LIN {X 0,Y 64.244,Z 442.937,A -85,B 0,C 180,E1 -28515.759,E2 -28515.759} C_VEL
LIN {X 0,Y 63.406,Z 448.254,A -85,B 0,C 180,E1 -28523.644,E2 -28523.644} C_VEL
LIN {X 0,Y 63.515,Z 451.726,A -85,B 0,C 180,E1 -28530.008,E2 -28530.008} C_VEL
LIN {X 0,Y 63.381,Z 454.429,A -85,B 0,C 180,E1 -28536.374,E2 -28536.374} C_VEL
LIN {X 0,Y 63.772,Z 456.467,A -85,B 0,C 180,E1 -28542.741,E2 -28542.741} C_VEL
LIN {X 0,Y 64.939,Z 458.028,A -85,B 0,C 180,E1 -28548.954,E2 -28548.954} C_VEL
LIN {X 0,Y 66.859,Z 459.178,A -85,B 0,C 180,E1 -28554.872,E2 -28554.872} C_VEL
LIN {X 0,Y 69.441,Z 459.905,A -85,B 0,C 180,E1 -28560.409,E2 -28560.409} C_VEL
LIN {X 0,Y 72.688,Z 460.091,A -85,B 0,C 180,E1 -28565.468,E2 -28565.468} C_VEL
LIN {X 0,Y 80.971,Z 459.289,A -85,B 0,C 180,E1 -28573.985,E2 -28573.985} C_VEL
LIN {X 0,Y 85.695,Z 458.239,A -85,B 0,C 180,E1 -28577.579,E2 -28577.579} C_VEL
LIN {X 0,Y 90.746,Z 456.64,A -85,B 0,C 180,E1 -28580.765,E2 -28580.765} C_VEL
LIN {X 0,Y 95.673,Z 454.631,A -85,B 0,C 180,E1 -28584.004,E2 -28584.004} C_VEL
LIN {X 0,Y 97.875,Z 453.563,A -85,B 0,C 180,E1 -28585.671,E2 -28585.671} C_VEL
LIN {X 0,Y 99.222,Z 452.513,A -85,B 0,C 180,E1 -28588.217,E2 -28588.217} C_VEL
LIN {X 0,Y 99.958,Z 451.651,A -85,B 0,C 180,E1 -28590.513,E2 -28590.513} C_VEL
LIN {X 0,Y 100.672,Z 450.423,A -85,B 0,C 180,E1 -28595.233,E2 -28595.233} C_VEL
LIN {X 0,Y 101.17,Z 449.63,A -85,B 0,C 180,E1 -28599.672,E2 -28599.672} C_VEL
LIN {X 0,Y 101.648,Z 449.123,A -85,B 0,C 180,E1 -28605.476,E2 -28605.476} C_VEL
LIN {X 0,Y 101.76,Z 449.101,A -85,B 0,C 180,E1 -28608.038,E2 -28608.038} C_VEL
LIN {X 0,Y 101.473,Z 449.465,A -85,B 0,C 180,E1 -28612.034,E2 -28612.034} C_VEL
LIN {X 0,Y 100.225,Z 450.423,A -85,B 0,C 180,E1 -28615.975,E2 -28615.975} C_VEL
LIN {X 0,Y 98.443,Z 451.251,A -85,B 0,C 180,E1 -28618.299,E2 -28618.299} C_VEL
LIN {X 0,Y 91.433,Z 453.624,A -85,B 0,C 180,E1 -28622.083,E2 -28622.083} C_VEL
LIN {X 0,Y 84.871,Z 455.149,A -85,B 0,C 180,E1 -28626.388,E2 -28626.388} C_VEL
LIN {X 0,Y 78.872,Z 455.858,A -85,B 0,C 180,E1 -28631.4,E2 -28631.4} C_VEL
LIN {X 0,Y 73.6,Z 455.754,A -85,B 0,C 180,E1 -28637.252,E2 -28637.252} C_VEL
LIN {X 0,Y 69.109,Z 454.82,A -85,B 0,C 180,E1 -28643.996,E2 -28643.996} C_VEL
LIN {X 0,Y 64.32,Z 451.791,A -85,B 0,C 180,E1 -28655.889,E2 -28655.889} C_VEL
LIN {X 0,Y 62.729,Z 448.38,A -85,B 0,C 180,E1 -28664.779,E2 -28664.779} C_VEL
LIN {X 0,Y 62.587,Z 443.781,A -85,B 0,C 180,E1 -28673.927,E2 -28673.927} C_VEL
LIN {X 0,Y 63.626,Z 438.495,A -85,B 0,C 180,E1 -28682.073,E2 -28682.073} C_VEL
LIN {X 0,Y 65.033,Z 433.873,A -85,B 0,C 180,E1 -28687.767,E2 -28687.767} C_VEL
LIN {X 0,Y 67.018,Z 428.034,A -85,B 0,C 180,E1 -28693.547,E2 -28693.547} C_VEL
LIN {X 0,Y 69.631,Z 420.592,A -85,B 0,C 180,E1 -28699.279,E2 -28699.279} C_VEL
LIN {X 0,Y 71.829,Z 414.232,A -85,B 0,C 180,E1 -28703.141,E2 -28703.141} C_VEL
LIN {X 0,Y 71.986,Z 407.933,A -85,B 0,C 180,E1 -28706.877,E2 -28706.877} C_VEL
LIN {X 0,Y 71.696,Z 402.285,A -85,B 0,C 180,E1 -28709.993,E2 -28709.993} C_VEL
LIN {X 0,Y 70.155,Z 394.65,A -85,B 0,C 180,E1 -28714.159,E2 -28714.159} C_VEL
LIN {X 0,Y 65.944,Z 385.726,A -85,B 0,C 180,E1 -28719.965,E2 -28719.965} C_VEL
LIN {X 0,Y 65.843,Z 385.09,A -85,B 0,C 180,E1 -28720.369,E2 -28720.369} C_VEL
LIN {X 0,Y 65.627,Z 385.123,A -85,B 0,C 180,E1 -28725.487,E2 -28725.487} C_VEL
LIN {X 0,Y 65.237,Z 385.169,A -85,B 0,C 180,E1 -28735.517,E2 -28735.517} C_VEL
LIN {X 0,Y 65.249,Z 385.167,A -85,B 0,C 180,E1 -28740.477,E2 -28740.477} C_VEL
LIN {X 0,Y 65.056,Z 385.207,A -85,B 0,C 180,E1 -28743.912,E2 -28743.912} C_VEL
LIN {X 0,Y 64.301,Z 385.311,A -85,B 0,C 180,E1 -28747.324,E2 -28747.324} C_VEL
LIN {X 0,Y 62.55,Z 385.533,A -85,B 0,C 180,E1 -28752.478,E2 -28752.478} C_VEL
LIN {X 0,Y 58.456,Z 386.017,A -85,B 0,C 180,E1 -28765.63,E2 -28765.63} C_VEL
LIN {X 0,Y 58.13,Z 386.048,A -85,B 0,C 180,E1 -28769.694,E2 -28769.694} C_VEL
LIN {X 0,Y 58.195,Z 386.04,A -85,B 0,C 180,E1 -28778.766,E2 -28778.766} C_VEL
LIN {X 0,Y 58.666,Z 385.984,A -85,B 0,C 180,E1 -28786.145,E2 -28786.145} C_VEL
LIN {X 0,Y 58.82,Z 385.97,A -85,B 0,C 180,E1 -28793.145,E2 -28793.145} C_VEL
LIN {X 0,Y 59.387,Z 385.901,A -85,B 0,C 180,E1 -28800.007,E2 -28800.007} C_VEL
LIN {X 0,Y 58.813,Z 385.969,A -85,B 0,C 180,E1 -28806.87,E2 -28806.87} C_VEL
LIN {X 0,Y 58.519,Z 386.008,A -85,B 0,C 180,E1 -28816.133,E2 -28816.133} C_VEL
LIN {X 0,Y 58.149,Z 386.046,A -85,B 0,C 180,E1 -28828.918,E2 -28828.918} C_VEL
LIN {X 0,Y 58.202,Z 386.231,A -85,B 0,C 180,E1 -28833.217,E2 -28833.217} C_VEL
LIN {X 0,Y 59.233,Z 388.945,A -85,B 0,C 180,E1 -28835.019,E2 -28835.019} C_VEL
LIN {X 0,Y 60.899,Z 391.865,A -85,B 0,C 180,E1 -28837.299,E2 -28837.299} C_VEL
LIN {X 0,Y 64.111,Z 398.641,A -85,B 0,C 180,E1 -28842.186,E2 -28842.186} C_VEL
LIN {X 0,Y 64.048,Z 403.218,A -85,B 0,C 180,E1 -28844.389,E2 -28844.389} C_VEL
LIN {X 0,Y 63.359,Z 410.92,A -85,B 0,C 180,E1 -28848.288,E2 -28848.288} C_VEL
LIN {X 0,Y 62.507,Z 418.749,A -85,B 0,C 180,E1 -28853.06,E2 -28853.06} C_VEL
LIN {X 0,Y 61.459,Z 426.817,A -85,B 0,C 180,E1 -28859.04,E2 -28859.04} C_VEL
LIN {X 0,Y 60.725,Z 430.806,A -85,B 0,C 180,E1 -28862.433,E2 -28862.433} C_VEL
LIN {X 0,Y 58.584,Z 437.173,A -85,B 0,C 180,E1 -28868.916,E2 -28868.916} C_VEL
LIN {X 0,Y 57.155,Z 442.475,A -85,B 0,C 180,E1 -28875.773,E2 -28875.773} C_VEL
LIN {X 0,Y 56.419,Z 446.887,A -85,B 0,C 180,E1 -28882.854,E2 -28882.854} C_VEL
LIN {X 0,Y 56.487,Z 450.536,A -85,B 0,C 180,E1 -28890.009,E2 -28890.009} C_VEL
LIN {X 0,Y 56.563,Z 454.501,A -85,B 0,C 180,E1 -28900.751,E2 -28900.751} C_VEL
LIN {X 0,Y 58.299,Z 457.233,A -85,B 0,C 180,E1 -28911.211,E2 -28911.211} C_VEL
LIN {X 0,Y 60.505,Z 458.548,A -85,B 0,C 180,E1 -28917.695,E2 -28917.695} C_VEL
LIN {X 0,Y 63.414,Z 459.31,A -85,B 0,C 180,E1 -28923.66,E2 -28923.66} C_VEL
LIN {X 0,Y 67.033,Z 459.66,A -85,B 0,C 180,E1 -28928.99,E2 -28928.99} C_VEL
LIN {X 0,Y 71.302,Z 459.641,A -85,B 0,C 180,E1 -28933.637,E2 -28933.637} C_VEL
LIN {X 0,Y 76.013,Z 459.192,A -85,B 0,C 180,E1 -28937.712,E2 -28937.712} C_VEL
LIN {X 0,Y 86.391,Z 456.813,A -85,B 0,C 180,E1 -28944.45,E2 -28944.45} C_VEL
LIN {X 0,Y 91.498,Z 455.061,A -85,B 0,C 180,E1 -28947.673,E2 -28947.673} C_VEL
LIN {X 0,Y 93.556,Z 453.407,A -85,B 0,C 180,E1 -28953.205,E2 -28953.205} C_VEL
LIN {X 0,Y 94.314,Z 452.529,A -85,B 0,C 180,E1 -28958.121,E2 -28958.121} C_VEL
LIN {X 0,Y 94.934,Z 451.878,A -85,B 0,C 180,E1 -28964.254,E2 -28964.254} C_VEL
LIN {X 0,Y 95.125,Z 451.749,A -85,B 0,C 180,E1 -28967.19,E2 -28967.19} C_VEL
LIN {X 0,Y 94.846,Z 451.894,A -85,B 0,C 180,E1 -28971.473,E2 -28971.473} C_VEL
LIN {X 0,Y 92.779,Z 452.842,A -85,B 0,C 180,E1 -28975.651,E2 -28975.651} C_VEL
LIN {X 0,Y 84.344,Z 455.086,A -85,B 0,C 180,E1 -28980.083,E2 -28980.083} C_VEL
LIN {X 0,Y 76.714,Z 456.16,A -85,B 0,C 180,E1 -28985.251,E2 -28985.251} C_VEL
LIN {X 0,Y 69.812,Z 456.21,A -85,B 0,C 180,E1 -28991.609,E2 -28991.609} C_VEL
LIN {X 0,Y 63.974,Z 455.229,A -85,B 0,C 180,E1 -28999.236,E2 -28999.236} C_VEL
LIN {X 0,Y 61.415,Z 454.386,A -85,B 0,C 180,E1 -29003.706,E2 -29003.706} C_VEL
LIN {X 0,Y 58.049,Z 452.174,A -85,B 0,C 180,E1 -29012.044,E2 -29012.044} C_VEL
LIN {X 0,Y 56.011,Z 449.085,A -85,B 0,C 180,E1 -29021.149,E2 -29021.149} C_VEL
LIN {X 0,Y 55.387,Z 445.043,A -85,B 0,C 180,E1 -29030.61,E2 -29030.61} C_VEL
LIN {X 0,Y 56.287,Z 439.309,A -85,B 0,C 180,E1 -29040.914,E2 -29040.914} C_VEL
LIN {X 0,Y 57.987,Z 433.695,A -85,B 0,C 180,E1 -29048.669,E2 -29048.669} C_VEL
LIN {X 0,Y 60.103,Z 427.827,A -85,B 0,C 180,E1 -29055.02,E2 -29055.02} C_VEL
LIN {X 0,Y 62.728,Z 420.854,A -85,B 0,C 180,E1 -29060.885,E2 -29060.885} C_VEL
LIN {X 0,Y 65.078,Z 414.476,A -85,B 0,C 180,E1 -29065.096,E2 -29065.096} C_VEL
LIN {X 0,Y 65.326,Z 406.891,A -85,B 0,C 180,E1 -29069.992,E2 -29069.992} C_VEL
LIN {X 0,Y 64.63,Z 400.768,A -85,B 0,C 180,E1 -29073.867,E2 -29073.867} C_VEL
LIN {X 0,Y 63.641,Z 396.893,A -85,B 0,C 180,E1 -29076.404,E2 -29076.404} C_VEL
LIN {X 0,Y 60.474,Z 389.846,A -85,B 0,C 180,E1 -29081.724,E2 -29081.724} C_VEL
LIN {X 0,Y 58.729,Z 386.66,A -85,B 0,C 180,E1 -29084.516,E2 -29084.516} C_VEL
LIN {X 0,Y 58.588,Z 385.999,A -85,B 0,C 180,E1 -29085.062,E2 -29085.062} C_VEL
LIN {X 0,Y 58.183,Z 386.043,A -85,B 0,C 180,E1 -29091.236,E2 -29091.236} C_VEL
LIN {X 0,Y 58.13,Z 386.049,A -85,B 0,C 180,E1 -29100.5,E2 -29100.5} C_VEL
LIN {X 0,Y 58.072,Z 386.056,A -85,B 0,C 180,E1 -29107.225,E2 -29107.225} C_VEL
LIN {X 0,Y 58.096,Z 386.056,A -85,B 0,C 180,E1 -29116.525,E2 -29116.525} C_VEL
LIN {X 0,Y 58.072,Z 386.055,A -85,B 0,C 180,E1 -29122.772,E2 -29122.772} C_VEL
LIN {X 0,Y 58.13,Z 386.048,A -85,B 0,C 180,E1 -29129.694,E2 -29129.694} C_VEL
LIN {X 0,Y 57.457,Z 386.138,A -85,B 0,C 180,E1 -29133.504,E2 -29133.504} C_VEL
LIN {X 0,Y 55.32,Z 386.4,A -85,B 0,C 180,E1 -29138.446,E2 -29138.446} C_VEL
LIN {X 0,Y 52.021,Z 386.813,A -85,B 0,C 180,E1 -29146.503,E2 -29146.503} C_VEL
LIN {X 0,Y 51.603,Z 386.862,A -85,B 0,C 180,E1 -29151.001,E2 -29151.001} C_VEL
LIN {X 0,Y 52.272,Z 386.787,A -85,B 0,C 180,E1 -29160.008,E2 -29160.008} C_VEL
LIN {X 0,Y 51.687,Z 386.859,A -85,B 0,C 180,E1 -29167.822,E2 -29167.822} C_VEL
LIN {X 0,Y 51.387,Z 386.897,A -85,B 0,C 180,E1 -29176.827,E2 -29176.827} C_VEL
LIN {X 0,Y 51.014,Z 386.94,A -85,B 0,C 180,E1 -29186.607,E2 -29186.607} C_VEL
LIN {X 0,Y 51.69,Z 389.043,A -85,B 0,C 180,E1 -29188.425,E2 -29188.425} C_VEL
LIN {X 0,Y 54.931,Z 394.782,A -85,B 0,C 180,E1 -29194.418,E2 -29194.418} C_VEL
LIN {X 0,Y 57.815,Z 401.379,A -85,B 0,C 180,E1 -29199.935,E2 -29199.935} C_VEL
LIN {X 0,Y 57.484,Z 406.739,A -85,B 0,C 180,E1 -29202.828,E2 -29202.828} C_VEL
LIN {X 0,Y 56.076,Z 416.989,A -85,B 0,C 180,E1 -29209.335,E2 -29209.335} C_VEL
LIN {X 0,Y 54.82,Z 425.167,A -85,B 0,C 180,E1 -29215.895,E2 -29215.895} C_VEL
LIN {X 0,Y 53.866,Z 430.299,A -85,B 0,C 180,E1 -29220.719,E2 -29220.719} C_VEL
LIN {X 0,Y 51.564,Z 436.691,A -85,B 0,C 180,E1 -29227.998,E2 -29227.998} C_VEL
LIN {X 0,Y 49.795,Z 443.14,A -85,B 0,C 180,E1 -29237.788,E2 -29237.788} C_VEL
LIN {X 0,Y 49.383,Z 448.166,A -85,B 0,C 180,E1 -29247.763,E2 -29247.763} C_VEL
LIN {X 0,Y 49.467,Z 451.386,A -85,B 0,C 180,E1 -29255.925,E2 -29255.925} C_VEL
LIN {X 0,Y 50.13,Z 454.494,A -85,B 0,C 180,E1 -29266.294,E2 -29266.294} C_VEL
LIN {X 0,Y 51.777,Z 456.418,A -85,B 0,C 180,E1 -29274.04,E2 -29274.04} C_VEL
LIN {X 0,Y 54.334,Z 457.781,A -85,B 0,C 180,E1 -29281.168,E2 -29281.168} C_VEL
LIN {X 0,Y 61.681,Z 459.227,A -85,B 0,C 180,E1 -29293.14,E2 -29293.14} C_VEL
LIN {X 0,Y 66.348,Z 459.371,A -85,B 0,C 180,E1 -29297.869,E2 -29297.869} C_VEL
LIN {X 0,Y 76.83,Z 458.172,A -85,B 0,C 180,E1 -29305.425,E2 -29305.425} C_VEL
LIN {X 0,Y 82.431,Z 456.99,A -85,B 0,C 180,E1 -29308.506,E2 -29308.506} C_VEL
LIN {X 0,Y 85.279,Z 456.105,A -85,B 0,C 180,E1 -29310.36,E2 -29310.36} C_VEL
LIN {X 0,Y 86.491,Z 455.449,A -85,B 0,C 180,E1 -29313.37,E2 -29313.37} C_VEL
LIN {X 0,Y 87.166,Z 454.978,A -85,B 0,C 180,E1 -29316.221,E2 -29316.221} C_VEL
LIN {X 0,Y 88.046,Z 454.174,A -85,B 0,C 180,E1 -29323.327,E2 -29323.327} C_VEL
LIN {X 0,Y 88.277,Z 454.004,A -85,B 0,C 180,E1 -29326.178,E2 -29326.178} C_VEL
LIN {X 0,Y 87.999,Z 453.998,A -85,B 0,C 180,E1 -29330.804,E2 -29330.804} C_VEL
LIN {X 0,Y 84.847,Z 454.764,A -85,B 0,C 180,E1 -29333.758,E2 -29333.758} C_VEL
LIN {X 0,Y 77.379,Z 456.109,A -85,B 0,C 180,E1 -29337.687,E2 -29337.687} C_VEL
LIN {X 0,Y 70.35,Z 456.651,A -85,B 0,C 180,E1 -29342.409,E2 -29342.409} C_VEL
LIN {X 0,Y 63.913,Z 456.399,A -85,B 0,C 180,E1 -29348.192,E2 -29348.192} C_VEL
LIN {X 0,Y 58.275,Z 455.348,A -85,B 0,C 180,E1 -29355.213,E2 -29355.213} C_VEL
LIN {X 0,Y 51.829,Z 452.306,A -85,B 0,C 180,E1 -29368.169,E2 -29368.169} C_VEL
LIN {X 0,Y 49.213,Z 448.934,A -85,B 0,C 180,E1 -29378.829,E2 -29378.829} C_VEL
LIN {X 0,Y 48.329,Z 444.335,A -85,B 0,C 180,E1 -29390.538,E2 -29390.538} C_VEL
LIN {X 0,Y 48.933,Z 439.98,A -85,B 0,C 180,E1 -29399.496,E2 -29399.496} C_VEL
LIN {X 0,Y 50.725,Z 434.072,A -85,B 0,C 180,E1 -29408.971,E2 -29408.971} C_VEL
LIN {X 0,Y 53.544,Z 426.81,A -85,B 0,C 180,E1 -29417.675,E2 -29417.675} C_VEL
LIN {X 0,Y 56.512,Z 419.546,A -85,B 0,C 180,E1 -29424.133,E2 -29424.133} C_VEL
LIN {X 0,Y 58.383,Z 414.861,A -85,B 0,C 180,E1 -29427.404,E2 -29427.404} C_VEL
LIN {X 0,Y 58.778,Z 407.72,A -85,B 0,C 180,E1 -29432.564,E2 -29432.564} C_VEL
LIN {X 0,Y 58.111,Z 401.727,A -85,B 0,C 180,E1 -29436.937,E2 -29436.937} C_VEL
LIN {X 0,Y 54.923,Z 393.934,A -85,B 0,C 180,E1 -29443.871,E2 -29443.871} C_VEL
LIN {X 0,Y 53.275,Z 390.905,A -85,B 0,C 180,E1 -29446.974,E2 -29446.974} C_VEL
LIN {X 0,Y 52.039,Z 389.44,A -85,B 0,C 180,E1 -29449.051,E2 -29449.051} C_VEL
LIN {X 0,Y 51.093,Z 386.927,A -85,B 0,C 180,E1 -29451.698,E2 -29451.698} C_VEL
LIN {X 0,Y 51.046,Z 386.934,A -85,B 0,C 180,E1 -29464.317,E2 -29464.317} C_VEL
LIN {X 0,Y 51.061,Z 386.93,A -85,B 0,C 180,E1 -29473.474,E2 -29473.474} C_VEL
LIN {X 0,Y 51.06,Z 386.931,A -85,B 0,C 180,E1 -29476.523,E2 -29476.523} C_VEL
LIN {X 0,Y 51.068,Z 386.936,A -85,B 0,C 180,E1 -29486.61,E2 -29486.61} C_VEL
LIN {X 0,Y 51.024,Z 386.942,A -85,B 0,C 180,E1 -29495.602,E2 -29495.602} C_VEL
LIN {X 0,Y 51.494,Z 386.883,A -85,B 0,C 180,E1 -29504.168,E2 -29504.168} C_VEL
LIN {X 0,Y 51.603,Z 386.862,A -85,B 0,C 180,E1 -29511.001,E2 -29511.001} C_VEL
LIN {X 0,Y 51.262,Z 386.917,A -85,B 0,C 180,E1 -29514.547,E2 -29514.547} C_VEL
LIN {X 0,Y 49.517,Z 387.138,A -85,B 0,C 180,E1 -29519.369,E2 -29519.369} C_VEL
LIN {X 0,Y 44.45,Z 387.752,A -85,B 0,C 180,E1 -29532.418,E2 -29532.418} C_VEL
LIN {X 0,Y 44.22,Z 387.776,A -85,B 0,C 180,E1 -29535.112,E2 -29535.112} C_VEL
LIN {X 0,Y 44.236,Z 387.931,A -85,B 0,C 180,E1 -29537.838,E2 -29537.838} C_VEL
LIN {X 0,Y 44.996,Z 390.576,A -85,B 0,C 180,E1 -29540.826,E2 -29540.826} C_VEL
LIN {X 0,Y 46.486,Z 392.608,A -85,B 0,C 180,E1 -29544.404,E2 -29544.404} C_VEL
LIN {X 0,Y 49.434,Z 398.739,A -85,B 0,C 180,E1 -29551.806,E2 -29551.806} C_VEL
LIN {X 0,Y 51.378,Z 403.395,A -85,B 0,C 180,E1 -29556.768,E2 -29556.768} C_VEL
LIN {X 0,Y 51.565,Z 404.776,A -85,B 0,C 180,E1 -29557.84,E2 -29557.84} C_VEL
LIN {X 0,Y 49.819,Z 415.66,A -85,B 0,C 180,E1 -29565.157,E2 -29565.157} C_VEL
LIN {X 0,Y 48.131,Z 424.486,A -85,B 0,C 180,E1 -29572.977,E2 -29572.977} C_VEL
LIN {X 0,Y 47.05,Z 429.707,A -85,B 0,C 180,E1 -29578.493,E2 -29578.493} C_VEL
LIN {X 0,Y 44.062,Z 437.49,A -85,B 0,C 180,E1 -29588.981,E2 -29588.981} C_VEL
LIN {X 0,Y 42.701,Z 442.579,A -85,B 0,C 180,E1 -29598.14,E2 -29598.14} C_VEL
LIN {X 0,Y 42.361,Z 446.724,A -85,B 0,C 180,E1 -29607.392,E2 -29607.392} C_VEL
LIN {X 0,Y 42.517,Z 450.282,A -85,B 0,C 180,E1 -29617.279,E2 -29617.279} C_VEL
LIN {X 0,Y 43.418,Z 453.483,A -85,B 0,C 180,E1 -29628.902,E2 -29628.902} C_VEL
LIN {X 0,Y 45.42,Z 455.468,A -85,B 0,C 180,E1 -29637.671,E2 -29637.671} C_VEL
LIN {X 0,Y 52.192,Z 458.051,A -85,B 0,C 180,E1 -29652.334,E2 -29652.334} C_VEL
LIN {X 0,Y 56.715,Z 458.769,A -85,B 0,C 180,E1 -29658.045,E2 -29658.045} C_VEL
LIN {X 0,Y 61.814,Z 458.954,A -85,B 0,C 180,E1 -29662.75,E2 -29662.75} C_VEL
LIN {X 0,Y 73.032,Z 458.144,A -85,B 0,C 180,E1 -29670.02,E2 -29670.02} C_VEL
LIN {X 0,Y 78.886,Z 457.108,A -85,B 0,C 180,E1 -29673,E2 -29673} C_VEL
LIN {X 0,Y 79.372,Z 456.964,A -85,B 0,C 180,E1 -29673.717,E2 -29673.717} C_VEL
LIN {X 0,Y 80.564,Z 456.193,A -85,B 0,C 180,E1 -29679.573,E2 -29679.573} C_VEL
LIN {X 0,Y 81.245,Z 455.725,A -85,B 0,C 180,E1 -29684.954,E2 -29684.954} C_VEL
LIN {X 0,Y 80.235,Z 455.81,A -85,B 0,C 180,E1 -29689.906,E2 -29689.906} C_VEL
LIN {X 0,Y 70.579,Z 456.928,A -85,B 0,C 180,E1 -29694.799,E2 -29694.799} C_VEL
LIN {X 0,Y 62.946,Z 456.972,A -85,B 0,C 180,E1 -29699.994,E2 -29699.994} C_VEL
LIN {X 0,Y 55.358,Z 456.013,A -85,B 0,C 180,E1 -29707.286,E2 -29707.286} C_VEL
LIN {X 0,Y 48.893,Z 454.004,A -85,B 0,C 180,E1 -29716.699,E2 -29716.699} C_VEL
LIN {X 0,Y 44.169,Z 450.918,A -85,B 0,C 180,E1 -29728.502,E2 -29728.502} C_VEL
LIN {X 0,Y 41.608,Z 446.616,A -85,B 0,C 180,E1 -29742.49,E2 -29742.49} C_VEL
LIN {X 0,Y 41.603,Z 440.621,A -85,B 0,C 180,E1 -29757.615,E2 -29757.615} C_VEL
LIN {X 0,Y 43.312,Z 434.893,A -85,B 0,C 180,E1 -29768.574,E2 -29768.574} C_VEL
LIN {X 0,Y 45.938,Z 428.413,A -85,B 0,C 180,E1 -29777.845,E2 -29777.845} C_VEL
LIN {X 0,Y 49.322,Z 420.79,A -85,B 0,C 180,E1 -29785.789,E2 -29785.789} C_VEL
LIN {X 0,Y 51.59,Z 415.524,A -85,B 0,C 180,E1 -29789.99,E2 -29789.99} C_VEL
LIN {X 0,Y 52.07,Z 412.568,A -85,B 0,C 180,E1 -29792.414,E2 -29792.414} C_VEL
LIN {X 0,Y 52.248,Z 407.816,A -85,B 0,C 180,E1 -29796.271,E2 -29796.271} C_VEL
LIN {X 0,Y 51.93,Z 404.62,A -85,B 0,C 180,E1 -29799.043,E2 -29799.043} C_VEL
LIN {X 0,Y 50.038,Z 399.481,A -85,B 0,C 180,E1 -29804.424,E2 -29804.424} C_VEL
LIN {X 0,Y 48.326,Z 395.727,A -85,B 0,C 180,E1 -29809.054,E2 -29809.054} C_VEL
LIN {X 0,Y 46.194,Z 392.128,A -85,B 0,C 180,E1 -29814.12,E2 -29814.12} C_VEL
LIN {X 0,Y 44.492,Z 389.97,A -85,B 0,C 180,E1 -29818.273,E2 -29818.273} C_VEL
LIN {X 0,Y 43.903,Z 387.827,A -85,B 0,C 180,E1 -29821.145,E2 -29821.145} C_VEL
LIN {X 0,Y 43.884,Z 387.83,A -85,B 0,C 180,E1 -29829.821,E2 -29829.821} C_VEL
LIN {X 0,Y 43.884,Z 387.822,A -85,B 0,C 180,E1 -29843.181,E2 -29843.181} C_VEL
LIN {X 0,Y 43.85,Z 387.826,A -85,B 0,C 180,E1 -29851.272,E2 -29851.272} C_VEL
LIN {X 0,Y 44.253,Z 387.782,A -85,B 0,C 180,E1 -29862.3,E2 -29862.3} C_VEL
LIN {X 0,Y 44.553,Z 387.745,A -85,B 0,C 180,E1 -29871.059,E2 -29871.059} C_VEL
LIN {X 0,Y 45.146,Z 387.674,A -85,B 0,C 180,E1 -29880.009,E2 -29880.009} C_VEL
LIN {X 0,Y 44.537,Z 387.75,A -85,B 0,C 180,E1 -29889.088,E2 -29889.088} C_VEL
LIN {X 0,Y 44.22,Z 387.776,A -85,B 0,C 180,E1 -29895.112,E2 -29895.112} C_VEL
LIN {X 0,Y 44.634,Z 388.607,A -85,B 0,C 180,E1 -29898.499,E2 -29898.499} C_VEL
LIN {X 0,Y 45.361,Z 391.009,A -85,B 0,C 180,E1 -29901.689,E2 -29901.689} C_VEL
LIN {X 0,Y 45.436,Z 394.448,A -85,B 0,C 180,E1 -29904.353,E2 -29904.353} C_VEL
LIN {X 0,Y 44.397,Z 402.478,A -85,B 0,C 180,E1 -29909.406,E2 -29909.406} C_VEL
LIN {X 0,Y 44.73,Z 404.749,A -85,B 0,C 180,E1 -29911.735,E2 -29911.735} C_VEL
LIN {X 0,Y 45.406,Z 406.963,A -85,B 0,C 180,E1 -29914.273,E2 -29914.273} C_VEL
LIN {X 0,Y 43.257,Z 416.646,A -85,B 0,C 180,E1 -29921.979,E2 -29921.979} C_VEL
LIN {X 0,Y 41.337,Z 424.824,A -85,B 0,C 180,E1 -29930.406,E2 -29930.406} C_VEL
LIN {X 0,Y 40.321,Z 429.037,A -85,B 0,C 180,E1 -29935.51,E2 -29935.51} C_VEL
LIN {X 0,Y 37.049,Z 436.89,A -85,B 0,C 180,E1 -29947.719,E2 -29947.719} C_VEL
LIN {X 0,Y 35.593,Z 442.01,A -85,B 0,C 180,E1 -29958.627,E2 -29958.627} C_VEL
LIN {X 0,Y 35.405,Z 446.282,A -85,B 0,C 180,E1 -29970.015,E2 -29970.015} C_VEL
LIN {X 0,Y 35.711,Z 449.682,A -85,B 0,C 180,E1 -29981.365,E2 -29981.365} C_VEL
LIN {X 0,Y 37.941,Z 453.437,A -85,B 0,C 180,E1 -29997.602,E2 -29997.602} C_VEL
LIN {X 0,Y 42.854,Z 456.111,A -85,B 0,C 180,E1 -30011.011,E2 -30011.011} C_VEL
LIN {X 0,Y 47.19,Z 457.4,A -85,B 0,C 180,E1 -30018.145,E2 -30018.145} C_VEL
LIN {X 0,Y 52.243,Z 458.161,A -85,B 0,C 180,E1 -30023.835,E2 -30023.835} C_VEL
LIN {X 0,Y 63.648,Z 458.507,A -85,B 0,C 180,E1 -30032.067,E2 -30032.067} C_VEL
LIN {X 0,Y 69.75,Z 458.066,A -85,B 0,C 180,E1 -30035.089,E2 -30035.089} C_VEL
LIN {X 0,Y 72.905,Z 457.545,A -85,B 0,C 180,E1 -30037.314,E2 -30037.314} C_VEL
LIN {X 0,Y 74.068,Z 456.99,A -85,B 0,C 180,E1 -30043.456,E2 -30043.456} C_VEL
LIN {X 0,Y 73.97,Z 456.901,A -85,B 0,C 180,E1 -30045.594,E2 -30045.594} C_VEL
LIN {X 0,Y 72.024,Z 457.104,A -85,B 0,C 180,E1 -30047.396,E2 -30047.396} C_VEL
LIN {X 0,Y 60.653,Z 457.348,A -85,B 0,C 180,E1 -30053.34,E2 -30053.34} C_VEL
LIN {X 0,Y 52.171,Z 456.393,A -85,B 0,C 180,E1 -30059.992,E2 -30059.992} C_VEL
LIN {X 0,Y 43.066,Z 453.794,A -85,B 0,C 180,E1 -30071.664,E2 -30071.664} C_VEL
LIN {X 0,Y 38.166,Z 450.911,A -85,B 0,C 180,E1 -30082.934,E2 -30082.934} C_VEL
LIN {X 0,Y 34.66,Z 445.941,A -85,B 0,C 180,E1 -30100.665,E2 -30100.665} C_VEL
LIN {X 0,Y 34.35,Z 441.216,A -85,B 0,C 180,E1 -30114.904,E2 -30114.904} C_VEL
LIN {X 0,Y 36.284,Z 434.569,A -85,B 0,C 180,E1 -30130.186,E2 -30130.186} C_VEL
LIN {X 0,Y 38.773,Z 428.997,A -85,B 0,C 180,E1 -30139.543,E2 -30139.543} C_VEL
LIN {X 0,Y 42.185,Z 421.994,A -85,B 0,C 180,E1 -30148.06,E2 -30148.06} C_VEL
LIN {X 0,Y 45.374,Z 415.138,A -85,B 0,C 180,E1 -30154.154,E2 -30154.154} C_VEL
LIN {X 0,Y 45.945,Z 410.355,A -85,B 0,C 180,E1 -30158.787,E2 -30158.787} C_VEL
LIN {X 0,Y 45.821,Z 407.812,A -85,B 0,C 180,E1 -30161.266,E2 -30161.266} C_VEL
LIN {X 0,Y 43.973,Z 402.105,A -85,B 0,C 180,E1 -30168.629,E2 -30168.629} C_VEL
LIN {X 0,Y 41.859,Z 397.763,A -85,B 0,C 180,E1 -30175.622,E2 -30175.622} C_VEL
LIN {X 0,Y 39.5,Z 393.395,A -85,B 0,C 180,E1 -30184.615,E2 -30184.615} C_VEL
LIN {X 0,Y 36.999,Z 390.172,A -85,B 0,C 180,E1 -30195.977,E2 -30195.977} C_VEL
LIN {X 0,Y 36.777,Z 388.714,A -85,B 0,C 180,E1 -30199.831,E2 -30199.831} C_VEL
LIN {X 0,Y 36.75,Z 388.713,A -85,B 0,C 180,E1 -30205.004,E2 -30205.004} C_VEL
LIN {X 0,Y 37.075,Z 388.672,A -85,B 0,C 180,E1 -30221.362,E2 -30221.362} C_VEL
LIN {X 0,Y 37.348,Z 388.637,A -85,B 0,C 180,E1 -30229.165,E2 -30229.165} C_VEL
LIN {X 0,Y 38.005,Z 388.564,A -85,B 0,C 180,E1 -30240.01,E2 -30240.01} C_VEL
LIN {X 0,Y 37.798,Z 388.715,A -85,B 0,C 180,E1 -30242.675,E2 -30242.675} C_VEL
LIN {X 0,Y 37.993,Z 390.234,A -85,B 0,C 180,E1 -30245.317,E2 -30245.317} C_VEL
LIN {X 0,Y 39.66,Z 393.158,A -85,B 0,C 180,E1 -30253.379,E2 -30253.379} C_VEL
LIN {X 0,Y 41.998,Z 397.914,A -85,B 0,C 180,E1 -30262.128,E2 -30262.128} C_VEL
LIN {X 0,Y 44.73,Z 404.749,A -85,B 0,C 180,E1 -30271.735,E2 -30271.735} C_VEL
LIN {X 0,Y 44.887,Z 406.8,A -85,B 0,C 180,E1 -30273.622,E2 -30273.622} C_VEL
LIN {X 0,Y 43.749,Z 410.066,A -85,B 0,C 180,E1 -30275.62,E2 -30275.62} C_VEL
LIN {X 0,Y 41.685,Z 413.338,A -85,B 0,C 180,E1 -30277.013,E2 -30277.013} C_VEL
LIN {X 0,Y 37.353,Z 418.963,A -85,B 0,C 180,E1 -30279.755,E2 -30279.755} C_VEL
LIN {X 0,Y 35.527,Z 422.293,A -85,B 0,C 180,E1 -30282.994,E2 -30282.994} C_VEL
LIN {X 0,Y 33.737,Z 428.341,A -85,B 0,C 180,E1 -30291.341,E2 -30291.341} C_VEL
LIN {X 0,Y 30.074,Z 436.258,A -85,B 0,C 180,E1 -30305.88,E2 -30305.88} C_VEL
LIN {X 0,Y 28.383,Z 442.279,A -85,B 0,C 180,E1 -30322.176,E2 -30322.176} C_VEL
LIN {X 0,Y 28.404,Z 444.726,A -85,B 0,C 180,E1 -30330.018,E2 -30330.018} C_VEL
LIN {X 0,Y 28.926,Z 448.229,A -85,B 0,C 180,E1 -30344.08,E2 -30344.08} C_VEL
LIN {X 0,Y 31.88,Z 452.324,A -85,B 0,C 180,E1 -30363.463,E2 -30363.463} C_VEL
LIN {X 0,Y 37.803,Z 455.26,A -85,B 0,C 180,E1 -30378.063,E2 -30378.063} C_VEL
LIN {X 0,Y 42.804,Z 456.588,A -85,B 0,C 180,E1 -30385.2,E2 -30385.2} C_VEL
LIN {X 0,Y 54.415,Z 458.075,A -85,B 0,C 180,E1 -30394.721,E2 -30394.721} C_VEL
LIN {X 0,Y 60.644,Z 458.222,A -85,B 0,C 180,E1 -30398.011,E2 -30398.011} C_VEL
LIN {X 0,Y 66.51,Z 457.817,A -85,B 0,C 180,E1 -30401.512,E2 -30401.512} C_VEL
LIN {X 0,Y 66.063,Z 457.741,A -85,B 0,C 180,E1 -30403.252,E2 -30403.252} C_VEL
LIN {X 0,Y 57.704,Z 457.618,A -85,B 0,C 180,E1 -30407.034,E2 -30407.034} C_VEL
LIN {X 0,Y 49.678,Z 456.714,A -85,B 0,C 180,E1 -30412.084,E2 -30412.084} C_VEL
LIN {X 0,Y 38.357,Z 453.784,A -85,B 0,C 180,E1 -30424.062,E2 -30424.062} C_VEL
LIN {X 0,Y 32.121,Z 450.514,A -85,B 0,C 180,E1 -30436.916,E2 -30436.916} C_VEL
LIN {X 0,Y 28.154,Z 446.1,A -85,B 0,C 180,E1 -30454.462,E2 -30454.462} C_VEL
LIN {X 0,Y 27.299,Z 440.438,A -85,B 0,C 180,E1 -30475.052,E2 -30475.052} C_VEL
LIN {X 0,Y 28.958,Z 434.957,A -85,B 0,C 180,E1 -30490.646,E2 -30490.646} C_VEL
LIN {X 0,Y 32.731,Z 427.411,A -85,B 0,C 180,E1 -30505.366,E2 -30505.366} C_VEL
LIN {X 0,Y 37.836,Z 418.104,A -85,B 0,C 180,E1 -30516.653,E2 -30516.653} C_VEL
LIN {X 0,Y 39.177,Z 415.325,A -85,B 0,C 180,E1 -30519.018,E2 -30519.018} C_VEL
LIN {X 0,Y 39.747,Z 411.198,A -85,B 0,C 180,E1 -30523.786,E2 -30523.786} C_VEL
LIN {X 0,Y 39.1,Z 408.116,A -85,B 0,C 180,E1 -30528.163,E2 -30528.163} C_VEL
LIN {X 0,Y 37.806,Z 404.538,A -85,B 0,C 180,E1 -30534.71,E2 -30534.71} C_VEL
LIN {X 0,Y 35.419,Z 399.011,A -85,B 0,C 180,E1 -30547.486,E2 -30547.486} C_VEL
LIN {X 0,Y 34.221,Z 397.497,A -85,B 0,C 180,E1 -30554.061,E2 -30554.061} C_VEL
LIN {X 0,Y 33.604,Z 395.517,A -85,B 0,C 180,E1 -30561.155,E2 -30561.155} C_VEL
LIN {X 0,Y 32.884,Z 394.747,A -85,B 0,C 180,E1 -30568.716,E2 -30568.716} C_VEL
LIN {X 0,Y 32.932,Z 394.275,A -85,B 0,C 180,E1 -30587.69,E2 -30587.69} C_VEL
LIN {X 0,Y 34.362,Z 395.335,A -85,B 0,C 180,E1 -30600.012,E2 -30600.012} C_VEL
LIN {X 0,Y 35.842,Z 399.216,A -85,B 0,C 180,E1 -30611.319,E2 -30611.319} C_VEL
LIN {X 0,Y 37.672,Z 404.304,A -85,B 0,C 180,E1 -30621.919,E2 -30621.919} C_VEL
LIN {X 0,Y 39.21,Z 408.896,A -85,B 0,C 180,E1 -30629.543,E2 -30629.543} C_VEL
LIN {X 0,Y 37.496,Z 415.574,A -85,B 0,C 180,E1 -30635.583,E2 -30635.583} C_VEL
LIN {X 0,Y 35.527,Z 422.293,A -85,B 0,C 180,E1 -30642.994,E2 -30642.994} C_VEL
LIN {X 0,Y 34.156,Z 425.306,A -85,B 0,C 180,E1 -30646.668,E2 -30646.668} C_VEL
LIN {X 0,Y 31.182,Z 429.496,A -85,B 0,C 180,E1 -30652.022,E2 -30652.022} C_VEL
LIN {X 0,Y 27.675,Z 433.145,A -85,B 0,C 180,E1 -30658.102,E2 -30658.102} C_VEL
LIN {X 0,Y 22.469,Z 438.862,A -85,B 0,C 180,E1 -30673.309,E2 -30673.309} C_VEL
LIN {X 0,Y 21.356,Z 442.088,A -85,B 0,C 180,E1 -30686.334,E2 -30686.334} C_VEL
LIN {X 0,Y 21.739,Z 445.042,A -85,B 0,C 180,E1 -30699.326,E2 -30699.326} C_VEL
LIN {X 0,Y 24.527,Z 449.76,A -85,B 0,C 180,E1 -30724.991,E2 -30724.991} C_VEL
LIN {X 0,Y 28.482,Z 452.281,A -85,B 0,C 180,E1 -30737.78,E2 -30737.78} C_VEL
LIN {X 0,Y 33.517,Z 454.219,A -85,B 0,C 180,E1 -30747.036,E2 -30747.036} C_VEL
LIN {X 0,Y 45.349,Z 456.85,A -85,B 0,C 180,E1 -30758.441,E2 -30758.441} C_VEL
LIN {X 0,Y 47.412,Z 457.093,A -85,B 0,C 180,E1 -30759.632,E2 -30759.632} C_VEL
LIN {X 0,Y 50.495,Z 457.396,A -85,B 0,C 180,E1 -30762.384,E2 -30762.384} C_VEL
LIN {X 0,Y 43.37,Z 456.202,A -85,B 0,C 180,E1 -30766.53,E2 -30766.53} C_VEL
LIN {X 0,Y 35.372,Z 453.997,A -85,B 0,C 180,E1 -30773.551,E2 -30773.551} C_VEL
LIN {X 0,Y 28.206,Z 450.924,A -85,B 0,C 180,E1 -30784.452,E2 -30784.452} C_VEL
LIN {X 0,Y 21.769,Z 445.657,A -85,B 0,C 180,E1 -30807.256,E2 -30807.256} C_VEL
LIN {X 0,Y 20.187,Z 440.305,A -85,B 0,C 180,E1 -30832.432,E2 -30832.432} C_VEL
LIN {X 0,Y 21.96,Z 434.619,A -85,B 0,C 180,E1 -30853.7,E2 -30853.7} C_VEL
LIN {X 0,Y 25.88,Z 427.833,A -85,B 0,C 180,E1 -30869.98,E2 -30869.98} C_VEL
LIN {X 0,Y 31.689,Z 418.518,A -85,B 0,C 180,E1 -30882.797,E2 -30882.797} C_VEL
LIN {X 0,Y 33.156,Z 415.875,A -85,B 0,C 180,E1 -30885.166,E2 -30885.166} C_VEL
LIN {X 0,Y 33.662,Z 413.803,A -85,B 0,C 180,E1 -30887.87,E2 -30887.87} C_VEL
LIN {X 0,Y 33.032,Z 410.087,A -85,B 0,C 180,E1 -30895.166,E2 -30895.166} C_VEL
LIN {X 0,Y 31.951,Z 407.089,A -85,B 0,C 180,E1 -30902.955,E2 -30902.955} C_VEL
LIN {X 0,Y 30.881,Z 404.052,A -85,B 0,C 180,E1 -30913.036,E2 -30913.036} C_VEL
LIN {X 0,Y 30.023,Z 401.492,A -85,B 0,C 180,E1 -30925.336,E2 -30925.336} C_VEL
LIN {X 0,Y 29.695,Z 401.048,A -85,B 0,C 180,E1 -30931.764,E2 -30931.764} C_VEL
LIN {X 0,Y 29.864,Z 400.781,A -85,B 0,C 180,E1 -30946.403,E2 -30946.403} C_VEL
LIN {X 0,Y 30.912,Z 402.262,A -85,B 0,C 180,E1 -30960.013,E2 -30960.013} C_VEL
LIN {X 0,Y 31.505,Z 404.025,A -85,B 0,C 180,E1 -30966.417,E2 -30966.417} C_VEL
LIN {X 0,Y 32.641,Z 408.954,A -85,B 0,C 180,E1 -30978.855,E2 -30978.855} C_VEL
LIN {X 0,Y 33.163,Z 411.125,A -85,B 0,C 180,E1 -30983.425,E2 -30983.425} C_VEL
LIN {X 0,Y 32.41,Z 414.141,A -85,B 0,C 180,E1 -30986.773,E2 -30986.773} C_VEL
LIN {X 0,Y 28.997,Z 423.108,A -85,B 0,C 180,E1 -30998.057,E2 -30998.057} C_VEL
LIN {X 0,Y 27.423,Z 427.476,A -85,B 0,C 180,E1 -31005.216,E2 -31005.216} C_VEL
LIN {X 0,Y 23.152,Z 435.542,A -85,B 0,C 180,E1 -31022.939,E2 -31022.939} C_VEL
LIN {X 0,Y 21.356,Z 442.088,A -85,B 0,C 180,E1 -31046.334,E2 -31046.334} C_VEL
LIN {X 0,Y 20.991,Z 443.724,A -85,B 0,C 180,E1 -31053.941,E2 -31053.941} C_VEL
LIN {X 0,Y 19.75,Z 445.467,A -85,B 0,C 180,E1 -31065.588,E2 -31065.588} C_VEL
LIN {X 0,Y 19.097,Z 448.121,A -85,B 0,C 180,E1 -31093.042,E2 -31093.042} C_VEL
LIN {X 0,Y 21.022,Z 449.393,A -85,B 0,C 180,E1 -31102.655,E2 -31102.655} C_VEL
LIN {X 0,Y 30.272,Z 453.121,A -85,B 0,C 180,E1 -31118.272,E2 -31118.272} C_VEL
LIN {X 0,Y 31.776,Z 453.483,A -85,B 0,C 180,E1 -31123.141,E2 -31123.141} C_VEL
LIN {X 0,Y 24.829,Z 450.772,A -85,B 0,C 180,E1 -31130.642,E2 -31130.642} C_VEL
LIN {X 0,Y 17.226,Z 446.269,A -85,B 0,C 180,E1 -31148.696,E2 -31148.696} C_VEL
LIN {X 0,Y 13.41,Z 441.409,A -85,B 0,C 180,E1 -31178.115,E2 -31178.115} C_VEL
LIN {X 0,Y 13.877,Z 436.569,A -85,B 0,C 180,E1 -31208.367,E2 -31208.367} C_VEL
LIN {X 0,Y 18.27,Z 429.564,A -85,B 0,C 180,E1 -31234.602,E2 -31234.602} C_VEL
LIN {X 0,Y 23.378,Z 422.588,A -85,B 0,C 180,E1 -31247.472,E2 -31247.472} C_VEL
LIN {X 0,Y 26.995,Z 417.457,A -85,B 0,C 180,E1 -31253.063,E2 -31253.063} C_VEL
LIN {X 0,Y 27.79,Z 415.797,A -85,B 0,C 180,E1 -31255.037,E2 -31255.037} C_VEL
LIN {X 0,Y 27.528,Z 413.729,A -85,B 0,C 180,E1 -31260.682,E2 -31260.682} C_VEL
LIN {X 0,Y 26.793,Z 410.282,A -85,B 0,C 180,E1 -31272.841,E2 -31272.841} C_VEL
LIN {X 0,Y 26.389,Z 407.546,A -85,B 0,C 180,E1 -31287.834,E2 -31287.834} C_VEL
LIN {X 0,Y 26.392,Z 407.076,A -85,B 0,C 180,E1 -31304.572,E2 -31304.572} C_VEL
LIN {X 0,Y 27.071,Z 408.736,A -85,B 0,C 180,E1 -31320.015,E2 -31320.015} C_VEL
LIN {X 0,Y 27.417,Z 412.098,A -85,B 0,C 180,E1 -31331.099,E2 -31331.099} C_VEL
LIN {X 0,Y 27.568,Z 413.462,A -85,B 0,C 180,E1 -31334.784,E2 -31334.784} C_VEL
LIN {X 0,Y 27.144,Z 415.134,A -85,B 0,C 180,E1 -31337.796,E2 -31337.796} C_VEL
LIN {X 0,Y 23.146,Z 423.275,A -85,B 0,C 180,E1 -31349.243,E2 -31349.243} C_VEL
LIN {X 0,Y 21.579,Z 426.569,A -85,B 0,C 180,E1 -31355.53,E2 -31355.53} C_VEL
LIN {X 0,Y 19.292,Z 430.12,A -85,B 0,C 180,E1 -31363.271,E2 -31363.271} C_VEL
LIN {X 0,Y 15.574,Z 436.167,A -85,B 0,C 180,E1 -31383.213,E2 -31383.213} C_VEL
LIN {X 0,Y 14.43,Z 441.173,A -85,B 0,C 180,E1 -31410.036,E2 -31410.036} C_VEL
LIN {X 0,Y 15.038,Z 443.572,A -85,B 0,C 180,E1 -31425.039,E2 -31425.039} C_VEL
LIN {X 0,Y 19.233,Z 448.406,A -85,B 0,C 180,E1 -31456.993,E2 -31456.993} C_VEL
LIN {X 0,Y 21.022,Z 449.393,A -85,B 0,C 180,E1 -31462.655,E2 -31462.655} C_VEL
LIN {X 0,Y 21.147,Z 449.536,A -85,B 0,C 180,E1 -31465.504,E2 -31465.504} C_VEL
LIN {X 0,Y 20.043,Z 449.15,A -85,B 0,C 180,E1 -31470.562,E2 -31470.562} C_VEL
LIN {X 0,Y 17.051,Z 447.765,A -85,B 0,C 180,E1 -31478.007,E2 -31478.007} C_VEL
LIN {X 0,Y 10.83,Z 444.097,A -85,B 0,C 180,E1 -31493.471,E2 -31493.471} C_VEL
LIN {X 0,Y 6.628,Z 440.062,A -85,B 0,C 180,E1 -31527.3,E2 -31527.3} C_VEL
LIN {X 0,Y 9.615,Z 432.643,A -85,B 0,C 180,E1 -31600.474,E2 -31600.474} C_VEL
LIN {X 0,Y 15.957,Z 425.702,A -85,B 0,C 180,E1 -31618.304,E2 -31618.304} C_VEL
LIN {X 0,Y 21.873,Z 418.475,A -85,B 0,C 180,E1 -31625.531,E2 -31625.531} C_VEL
LIN {X 0,Y 22.211,Z 417.119,A -85,B 0,C 180,E1 -31629.229,E2 -31629.229} C_VEL
LIN {X 0,Y 22.239,Z 414.783,A -85,B 0,C 180,E1 -31640.822,E2 -31640.822} C_VEL
LIN {X 0,Y 22.474,Z 413.22,A -85,B 0,C 180,E1 -31661.796,E2 -31661.796} C_VEL
LIN {X 0,Y 22.556,Z 413.805,A -85,B 0,C 180,E1 -31671.055,E2 -31671.055} C_VEL
LIN {X 0,Y 22.513,Z 415.26,A -85,B 0,C 180,E1 -31680.018,E2 -31680.018} C_VEL
LIN {X 0,Y 22.436,Z 416.214,A -85,B 0,C 180,E1 -31684.063,E2 -31684.063} C_VEL
LIN {X 0,Y 22.081,Z 417.147,A -85,B 0,C 180,E1 -31686.195,E2 -31686.195} C_VEL
LIN {X 0,Y 17.456,Z 424.427,A -85,B 0,C 180,E1 -31697.123,E2 -31697.123} C_VEL
LIN {X 0,Y 15.345,Z 427.588,A -85,B 0,C 180,E1 -31703.733,E2 -31703.733} C_VEL
LIN {X 0,Y 9.17,Z 434.876,A -85,B 0,C 180,E1 -31730.102,E2 -31730.102} C_VEL
LIN {X 0,Y 8.007,Z 440.887,A -85,B 0,C 180,E1 -31788.446,E2 -31788.446} C_VEL
LIN {X 0,Y 11.151,Z 444.369,A -85,B 0,C 180,E1 -31820.887,E2 -31820.887} C_VEL
LIN {X 0,Y 15.369,Z 446.861,A -85,B 0,C 180,E1 -31836.229,E2 -31836.229} C_VEL
LIN {X 0,Y 14.671,Z 446.403,A -85,B 0,C 180,E1 -31843.471,E2 -31843.471} C_VEL
LIN {X 0,Y 7.33,Z 441.032,A -85,B 0,C 180,E1 -31876.264,E2 -31876.264} C_VEL
LIN {X 0,Y 6.628,Z 440.062,A -85,B 0,C 180,E1 -31887.3,E2 -31887.3} C_VEL
LIN {X 0,Y 5.518,Z 437.803,A -85,B 0,C 180,E1 -31916.649,E2 -31916.649} C_VEL
LIN {X 0,Y 5.881,Z 433.735,A -85,B 0,C 180,E1 -31972.808,E2 -31972.808} C_VEL
LIN {X 0,Y 9.475,Z 429.275,A -85,B 0,C 180,E1 -32001.199,E2 -32001.199} C_VEL
LIN {X 0,Y 12.172,Z 426.359,A -85,B 0,C 180,E1 -32004.526,E2 -32004.526} C_VEL
LIN {X 0,Y 17.322,Z 420.677,A -85,B 0,C 180,E1 -32004.185,E2 -32004.185} C_VEL
LIN {X 0,Y 17.896,Z 419.393,A -85,B 0,C 180,E1 -32016.901,E2 -32016.901} C_VEL
LIN {X 0,Y 18.187,Z 419.09,A -85,B 0,C 180,E1 -32023.621,E2 -32023.621} C_VEL
LIN {X 0,Y 17.954,Z 419.745,A -85,B 0,C 180,E1 -32029.451,E2 -32029.451} C_VEL
LIN {X 0,Y 11.736,Z 427.187,A -85,B 0,C 180,E1 -32037.25,E2 -32037.25} C_VEL
LIN {X 0,Y 3.996,Z 434.141,A -85,B 0,C 180,E1 -32043.037,E2 -32043.037} C_VEL
LIN {X 0,Y 1.246,Z 436.1,A -85,B 0,C 180,E1 -32040.318,E2 -32040.318} C_VEL
LIN {X 0,Y 8.485,Z 429.835,A -85,B 0,C 180,E1 -32005.816,E2 -32005.816} C_VEL
LIN {X 0,Y 12.172,Z 426.359,A -85,B 0,C 180,E1 -32004.526,E2 -32004.526} C_VEL
LIN {X 0,Y 15.644,Z 427.711,A -85,B 0,C 180,E1 -32004.111,E2 -32004.111} C_VEL
LIN {X 0,Y 15.644,Z 600,A -85,B 0,C 180,E1 -32004.111,E2 -32004.111} C_VEL
LIN {X 0,Y 15.644,Z 600,A -85,B 0,C 180,E1 -32004.111,E2 -32004.111}

QRS_NEXT_CUT()

QRS_NEXT()
QRS_HOME()

END
